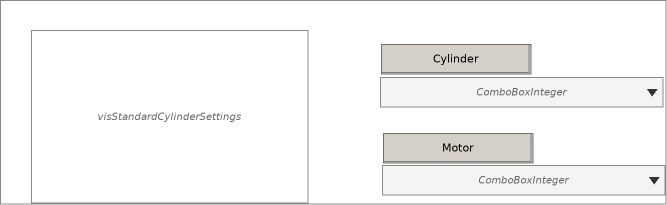
VISUALIZATION visSettingMachPart1  // 667x205
VAR_INPUT
	refSetting : REFERENCE TO ST_SettingMachinePart01;
END_VAR
VAR
	nSel : INT;
END_VAR
    Frame (31,30 277x173)
        shows visStandardCylinderSettings(refSetting := refSetting.stCylinderSettings)
        shows visStandardMotorSettings(refSetting := refSetting.stMotorSettings)
    Button (381,44 150x30), "Cylinder", colour toggle: nSel = 0
        OnMouseClick: FrameSelectionChange Selection=SelectedFrame=f571b872-985a-4510-9730-37c9a5269c7f, GlobSel=AssignType=Directly, SelType=Locally
        OnMouseClick: execute { nSel := 0; }
    Button (383,133 150x30), "Motor", colour toggle: nSel = 1
        OnMouseClick: FrameSelectionChange Selection=SelectedFrame=f571b872-985a-4510-9730-37c9a5269c7f, Selection=1, GlobSel=AssignType=Directly, SelType=Locally
        OnMouseClick: execute { nSel := 1; }
    ComboBoxInteger (380,77 283x30), variable: refSetting.nCylinderType, text list: 'txtCylinderTypes'
    ComboBoxInteger (382,165 283x30), variable: refSetting.nMotorType, text list: 'txtMotorTypes'
END_VISUALIZATION

(* stored: Version 1.1.0.1, ProductVersion 3.1.4019.2
   Visu visSettingMachPart1: Id {87e2958a-68a7-419e-9c5c-7bccdbc3cfd2} *)
